FUNCTION_BLOCK Fb_Motion
VAR_INPUT
END_VAR
VAR_OUTPUT
END_VAR
VAR
	mcPower: MC_Power;
	mcMoveAbs: MC_MoveAbsolute;
	mcStop: MC_Stop;
	McReset: MC_Reset;
END_VAR

VAR_IN_OUT
	
	Axis	:	AXIS_REF;
	stAxis	:	st_axisInterface;
	
END_VAR

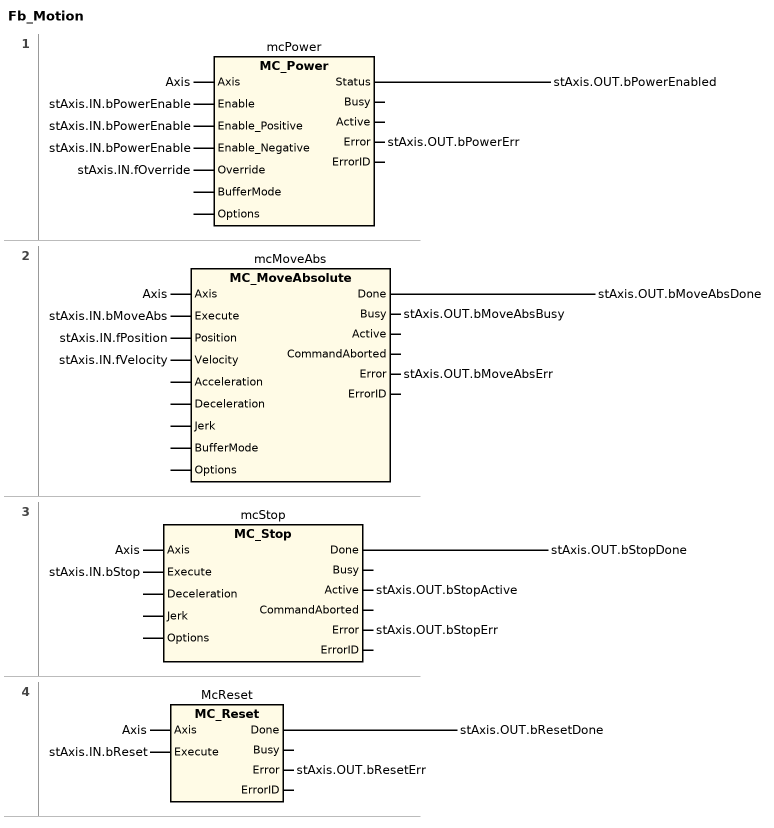
// NETWORK 1
mcPower(
    Axis := Axis,
    Enable := stAxis.IN.bPowerEnable,
    Enable_Positive := stAxis.IN.bPowerEnable,
    Enable_Negative := stAxis.IN.bPowerEnable,
    Override := stAxis.IN.fOverride,
    Error => stAxis.OUT.bPowerErr); // MC_Power
stAxis.OUT.bPowerEnabled := mcPower.Status;

// NETWORK 2
mcMoveAbs(
    Axis := Axis,
    Execute := stAxis.IN.bMoveAbs,
    Position := stAxis.IN.fPosition,
    Velocity := stAxis.IN.fVelocity,
    Busy => stAxis.OUT.bMoveAbsBusy,
    Error => stAxis.OUT.bMoveAbsErr); // MC_MoveAbsolute
stAxis.OUT.bMoveAbsDone := mcMoveAbs.Done;

// NETWORK 3
mcStop(
    Axis := Axis,
    Execute := stAxis.IN.bStop,
    Active => stAxis.OUT.bStopActive,
    Error => stAxis.OUT.bStopErr); // MC_Stop
stAxis.OUT.bStopDone := mcStop.Done;

// NETWORK 4
McReset(Axis := Axis, Execute := stAxis.IN.bReset, Error => stAxis.OUT.bResetErr); // MC_Reset
stAxis.OUT.bResetDone := McReset.Done;

END_FUNCTION_BLOCK

(* stored: Version 1.1.0.1, ProductVersion 3.1.4024.4
   POU Fb_Motion: Id {ebde0004-00c4-4d51-88a2-bdb9eda55382}, SpecialFunc None *)
